// TIA Portal V16 export
// export: Created 2024-05-14T12:25:18.4541934Z, ExportSetting WithDefaults, DisplayName Totally Integrated Automation Portal, DisplayVersion V16, DisplayName TIA Portal Version Control Interface, DisplayVersion V16, DisplayName TIA Portal Openness, DisplayVersion V16, DisplayName STEP 7 Professional, DisplayVersion V16, DisplayName STEP 7 Safety, DisplayVersion V16, DisplayName WinCC Advanced, DisplayVersion V16
FUNCTION_BLOCK "communicatie"   // FB12, LAD
{ S7_Optimized_Access := 'TRUE' }
VERSION : 0.1
// stored: AutoNumber true, IsIECCheckEnabled false, IsRetainMemResEnabled false, MemoryReserve 100, SetENOAutomatically false, UDAEnableTagReadback false
BEGIN

REGION Network 1
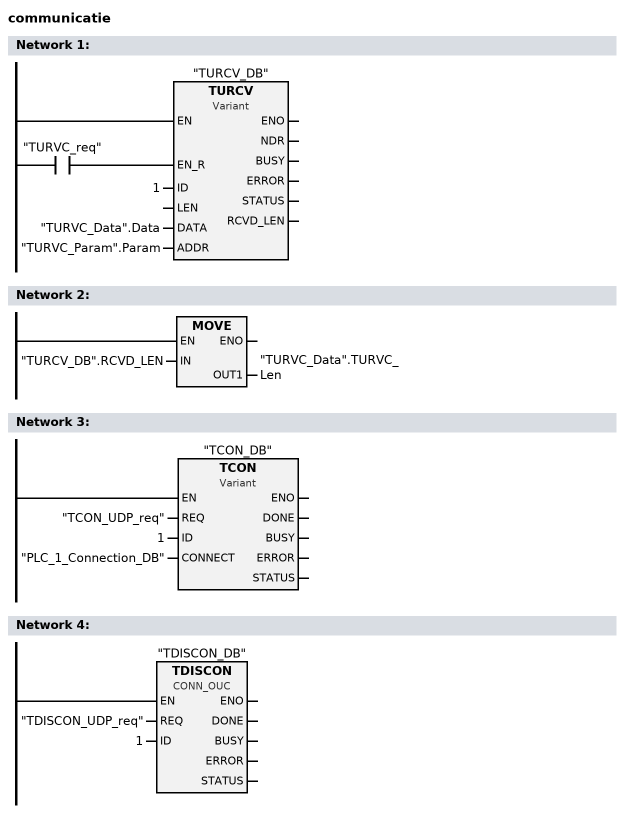
   RUNG wire#powerrail
      { S7_Templates := "[ptr_type := Variant, value_type := UDInt, id_type := CONN_OUC, addr_type := Variant]" } "TURCV_DB".TURCV(EN_R := wire#w1, ID := 1, LEN :=, DATA := "TURVC_Data".Data, ADDR := "TURVC_Param".Param, NDR =>, BUSY =>, ERROR =>, STATUS =>, RCVD_LEN =>)
   END_RUNG
   RUNG wire#powerrail
      Contact( "TURVC_req" )
   END_RUNG wire#w1
   // the same network as SCL:
   "TURCV_DB"(EN_R := "TURVC_req", ID := 1, DATA := "TURVC_Data".Data, ADDR := "TURVC_Param".Param);   // TURCV
END_REGION

REGION Network 2
   RUNG wire#powerrail
      Move(in := "TURCV_DB".RCVD_LEN, out1 => "TURVC_Data".TURVC_Len)
   END_RUNG
   // the same network as SCL:
   "TURVC_Data".TURVC_Len := "TURCV_DB".RCVD_LEN;
END_REGION

REGION Network 3
   RUNG wire#powerrail
      { S7_Templates := "[con_type := Variant, id_type := CONN_OUC]" } "TCON_DB".TCON(REQ := "TCON_UDP_req", ID := 1, CONNECT := "PLC_1_Connection_DB", DONE =>, BUSY =>, ERROR =>, STATUS =>)
   END_RUNG
   // the same network as SCL:
   "TCON_DB"(REQ := "TCON_UDP_req", ID := 1, CONNECT := "PLC_1_Connection_DB");   // TCON
END_REGION

REGION Network 4
   RUNG wire#powerrail
      { S7_Templates := "id_type := CONN_OUC" } "TDISCON_DB".TDISCON(REQ := "TDISCON_UDP_req", ID := 1, DONE =>, BUSY =>, ERROR =>, STATUS =>)
   END_RUNG
   // the same network as SCL:
   "TDISCON_DB"(REQ := "TDISCON_UDP_req", ID := 1);   // TDISCON
END_REGION
END_FUNCTION_BLOCK
